FUNCTION "LKinCtrl_RotZ" : Void
TITLE = LKinCtrl_RotZ
{ S7_Optimized_Access := 'TRUE' }
AUTHOR : 'handling.team.automation@siemens.com'
FAMILY : LKinCtrl
VERSION : 5.0
   VAR_INPUT
      angle : LReal;
   END_VAR

   VAR_IN_OUT
      rotMatrix : Array[1..3, 1..3] of LReal;
   END_VAR

   VAR_TEMP
      tempAngleRadians : LReal;
   END_VAR

   VAR CONSTANT
      PI : LReal := 3.14159265358979;   // Pi
   END_VAR


BEGIN
	// Rotationsmatrizen
	// RotZ:
	#tempAngleRadians := #angle * #PI / 180.0;

	// First row
	#rotMatrix[1, 1] := COS_LREAL(IN := #tempAngleRadians);
	#rotMatrix[1, 2] := - SIN_LREAL(IN := #tempAngleRadians);
	#rotMatrix[1, 3] := 0;

	// Second row
	#rotMatrix[2, 1] := SIN_LREAL(IN := #tempAngleRadians);
	#rotMatrix[2, 2] := COS_LREAL(IN := #tempAngleRadians);
	#rotMatrix[2, 3] := 0;

	// Third row
	#rotMatrix[3, 1] := 0;
	#rotMatrix[3, 2] := 0;
	#rotMatrix[3, 3] := 1;
END_FUNCTION

